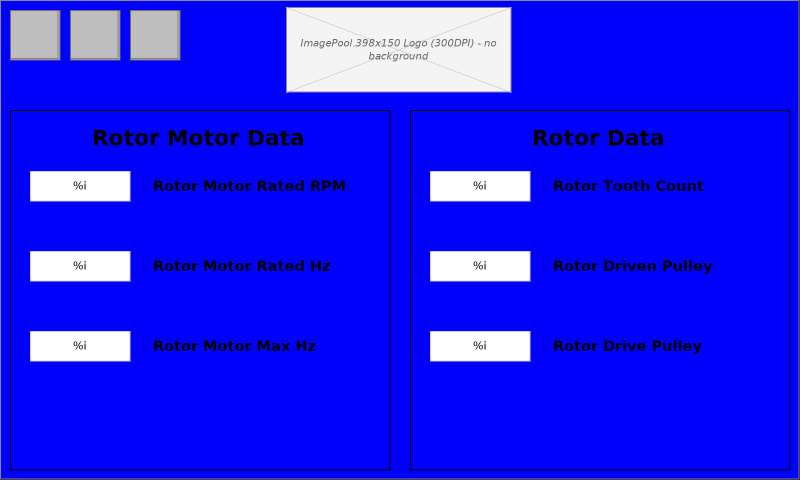
VISUALIZATION Rotor_Settings  // 800x480
    Rectangle (0,0 800x480)
    Rectangle (10,110 380x360)
    Textfield (30,171 100x30), "%i", text variable: GVL.RotorMot_Rated_RPM
        OnMouseClick: write the text variable via VisuDialogs.Numpad
    Rectangle (410,110 380x360)
    Textfield (30,251 100x30), "%i", text variable: GVL.RotorMot_Rated_Hz
        OnMouseClick: write the text variable via VisuDialogs.Numpad
    Textfield (30,331 100x30), "%i", text variable: GVL.RotorMot_Max_Hz
        OnMouseClick: write the text variable via VisuDialogs.Numpad
    Image (286,7 225x85), image: ImagePool.398x150 Logo (300DPI) - no background
        OnMouseClick: change screen: Home
    Button (70,10 50x50), image: VisuSymbols.Symbols.Home
        OnMouseClick: change screen: Home
    Label (20,120 357x36), "Rotor Motor Data"
    Label (420,120 357x36), "Rotor Data"
    Button (10,10 50x50), image: VisuSymbols.Symbols.TriangleLeft
        OnMouseClick: change screen: Previous Home
    Textfield (430,171 100x30), "%i", text variable: GVL.Rotor_Tooth_Count
        OnMouseClick: write the text variable via VisuDialogs.Numpad
    Textfield (430,251 100x30), "%i", text variable: GVL.Rotor_Driven_Pulley
        OnMouseClick: write the text variable via VisuDialogs.Numpad
    Textfield (430,331 100x30), "%i", text variable: GVL.Rotor_Drive_Pulley
        OnMouseClick: write the text variable via VisuDialogs.Numpad
    Label (150,171 225x30), "Rotor Motor Rated RPM"
    Label (150,251 225x30), "Rotor Motor Rated Hz"
    Label (150,331 225x30), "Rotor Motor Max Hz"
    Label (550,171 225x30), "Rotor Tooth Count"
    Label (550,251 225x30), "Rotor Driven Pulley"
    Label (550,331 225x30), "Rotor Drive Pulley"
    Button (130,10 50x50), image: VisuSymbols.Symbols.TwoWheels
        OnMouseClick: change screen: Settings_Menu
END_VISUALIZATION

(* stored: Version 1.1.0.1, ProductVersion 3.1.4024.12
   Visu Rotor_Settings: Id {eec97256-ef87-4a51-af8b-0f02d5fcfcd3} *)
